Staubli VAL3: GETFKEY.pgx

public program GetFKey(string x_sMenu, num& x_nSelect[])
  local string l_sMenuItm[8]
  local num l_nKey
  local bool l_bStop
begin
  // This routine returns the number of the function key pressed by the user
  // A menu item must be attached to the keypressed otherwise the routine
  // loops.
  //Convertion
  call _str2Array(x_sMenu," ",l_sMenuItm)
  l_nKey=getKey()
  // Function key has been pressed
  if (l_nKey>=271) and (l_nKey<=278)
    l_nKey=l_nKey-270
    l_nKey=sel(l_sMenuItm[l_nKey-1]!="",l_nKey,-1)
  endIf
  x_nSelect=l_nKey
end
